FUNCTION_BLOCK STEST_END (* Service Interface Function Block Type *)
  (* Standard: 61499-2 *)
  (* Version 1.0, 2015-01-11, Michael Hofmann, Profactor GmbH *)
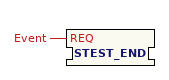
  EVENT_INPUT
    REQ; (* Service Request *)
  END_EVENT
  (* Service APPLICATION/RESOURCE: Service Interface Function Block Type *)
END_FUNCTION_BLOCK
(* other elements stored in the file *)
(* Identification Description=Copyright (c) 2015 Profactor GmbH This program and the accompanying materials are made available under the terms of the Eclipse Public License 2.0 which is available at https://www.eclipse.org/legal/epl-2.0/ SPDX-License-Identifier: EPL-2.0 *)
